// TIA Portal V18 export
FUNCTION "PLC8_910A1_CPU1214_IO_Update" : Void   // FC11010, LAD
{ S7_Optimized_Access := 'TRUE' }
VERSION : 0.1
// stored: AutoNumber false, IsIECCheckEnabled false, SetENOAutomatically false, UDAEnableTagReadback false
BEGIN

REGION Network 1: AI1 / "AI01.1.1" iw64
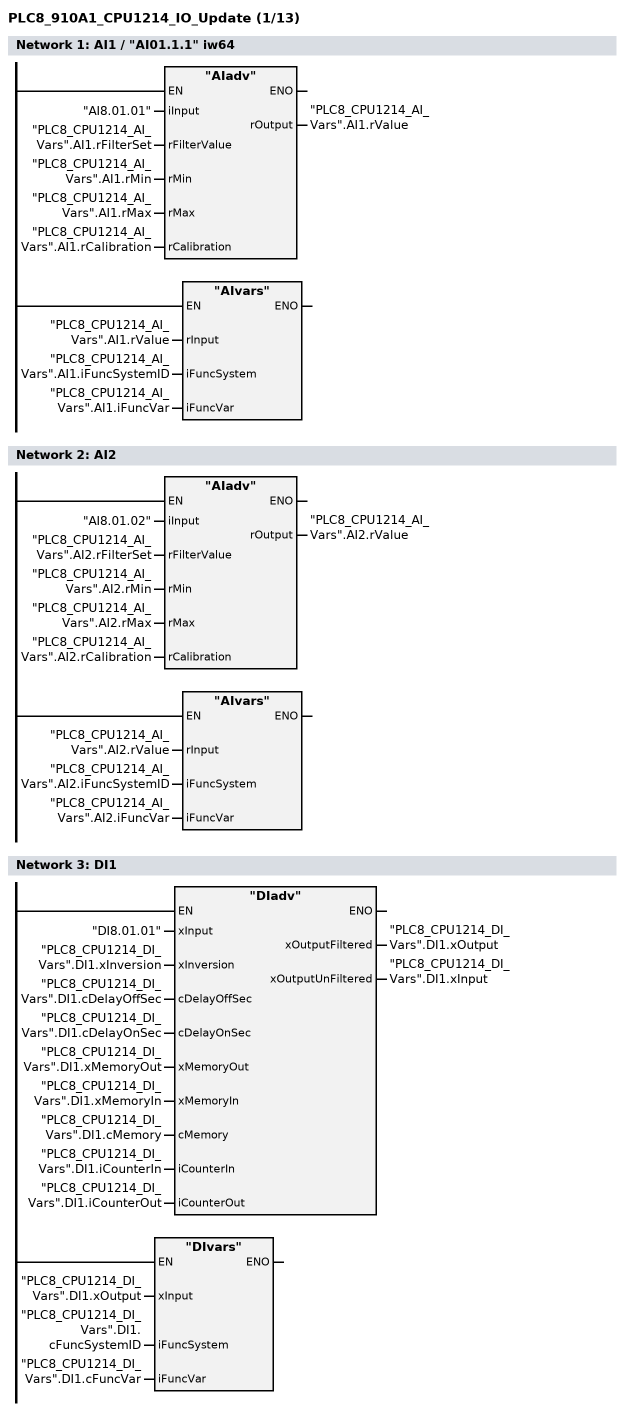
   RUNG wire#powerrail
      "AIadv"(iInput := "AI8.01.01", rFilterValue := "PLC8_CPU1214_AI_Vars".AI1.rFilterSet, rMin := "PLC8_CPU1214_AI_Vars".AI1.rMin, rMax := "PLC8_CPU1214_AI_Vars".AI1.rMax, rCalibration := "PLC8_CPU1214_AI_Vars".AI1.rCalibration, rOutput => "PLC8_CPU1214_AI_Vars".AI1.rValue)
   END_RUNG
   RUNG wire#powerrail
      "AIvars"(rInput := "PLC8_CPU1214_AI_Vars".AI1.rValue, iFuncSystem := "PLC8_CPU1214_AI_Vars".AI1.iFuncSystemID, iFuncVar := "PLC8_CPU1214_AI_Vars".AI1.iFuncVar)
   END_RUNG
   // the same network as SCL:
   "AIadv"(iInput := "AI8.01.01",
           rFilterValue := "PLC8_CPU1214_AI_Vars".AI1.rFilterSet,
           rMin := "PLC8_CPU1214_AI_Vars".AI1.rMin,
           rMax := "PLC8_CPU1214_AI_Vars".AI1.rMax,
           rCalibration := "PLC8_CPU1214_AI_Vars".AI1.rCalibration,
           rOutput => "PLC8_CPU1214_AI_Vars".AI1.rValue);
   "AIvars"(rInput := "PLC8_CPU1214_AI_Vars".AI1.rValue,
            iFuncSystem := "PLC8_CPU1214_AI_Vars".AI1.iFuncSystemID,
            iFuncVar := "PLC8_CPU1214_AI_Vars".AI1.iFuncVar);
END_REGION

REGION Network 2: AI2
   RUNG wire#powerrail
      "AIadv"(iInput := "AI8.01.02", rFilterValue := "PLC8_CPU1214_AI_Vars".AI2.rFilterSet, rMin := "PLC8_CPU1214_AI_Vars".AI2.rMin, rMax := "PLC8_CPU1214_AI_Vars".AI2.rMax, rCalibration := "PLC8_CPU1214_AI_Vars".AI2.rCalibration, rOutput => "PLC8_CPU1214_AI_Vars".AI2.rValue)
   END_RUNG
   RUNG wire#powerrail
      "AIvars"(rInput := "PLC8_CPU1214_AI_Vars".AI2.rValue, iFuncSystem := "PLC8_CPU1214_AI_Vars".AI2.iFuncSystemID, iFuncVar := "PLC8_CPU1214_AI_Vars".AI2.iFuncVar)
   END_RUNG
   // the same network as SCL:
   "AIadv"(iInput := "AI8.01.02",
           rFilterValue := "PLC8_CPU1214_AI_Vars".AI2.rFilterSet,
           rMin := "PLC8_CPU1214_AI_Vars".AI2.rMin,
           rMax := "PLC8_CPU1214_AI_Vars".AI2.rMax,
           rCalibration := "PLC8_CPU1214_AI_Vars".AI2.rCalibration,
           rOutput => "PLC8_CPU1214_AI_Vars".AI2.rValue);
   "AIvars"(rInput := "PLC8_CPU1214_AI_Vars".AI2.rValue,
            iFuncSystem := "PLC8_CPU1214_AI_Vars".AI2.iFuncSystemID,
            iFuncVar := "PLC8_CPU1214_AI_Vars".AI2.iFuncVar);
END_REGION

REGION Network 3: DI1
   RUNG wire#powerrail
      "DIadv"(xInput := "DI8.01.01", xInversion := "PLC8_CPU1214_DI_Vars".DI1.xInversion, cDelayOffSec := "PLC8_CPU1214_DI_Vars".DI1.cDelayOffSec, cDelayOnSec := "PLC8_CPU1214_DI_Vars".DI1.cDelayOnSec, xMemoryOut := "PLC8_CPU1214_DI_Vars".DI1.xMemoryOut, xMemoryIn := "PLC8_CPU1214_DI_Vars".DI1.xMemoryIn, cMemory := "PLC8_CPU1214_DI_Vars".DI1.cMemory, iCounterIn := "PLC8_CPU1214_DI_Vars".DI1.iCounterIn, iCounterOut := "PLC8_CPU1214_DI_Vars".DI1.iCounterOut, xOutputFiltered => "PLC8_CPU1214_DI_Vars".DI1.xOutput, xOutputUnFiltered => "PLC8_CPU1214_DI_Vars".DI1.xInput)
   END_RUNG
   RUNG wire#powerrail
      "DIvars"(xInput := "PLC8_CPU1214_DI_Vars".DI1.xOutput, iFuncSystem := "PLC8_CPU1214_DI_Vars".DI1.cFuncSystemID, iFuncVar := "PLC8_CPU1214_DI_Vars".DI1.cFuncVar)
   END_RUNG
   // the same network as SCL:
   "DIadv"(xInput := "DI8.01.01",
           xInversion := "PLC8_CPU1214_DI_Vars".DI1.xInversion,
           cDelayOffSec := "PLC8_CPU1214_DI_Vars".DI1.cDelayOffSec,
           cDelayOnSec := "PLC8_CPU1214_DI_Vars".DI1.cDelayOnSec,
           xMemoryOut := "PLC8_CPU1214_DI_Vars".DI1.xMemoryOut,
           xMemoryIn := "PLC8_CPU1214_DI_Vars".DI1.xMemoryIn,
           cMemory := "PLC8_CPU1214_DI_Vars".DI1.cMemory,
           iCounterIn := "PLC8_CPU1214_DI_Vars".DI1.iCounterIn,
           iCounterOut := "PLC8_CPU1214_DI_Vars".DI1.iCounterOut,
           xOutputFiltered => "PLC8_CPU1214_DI_Vars".DI1.xOutput,
           xOutputUnFiltered => "PLC8_CPU1214_DI_Vars".DI1.xInput);
   "DIvars"(xInput := "PLC8_CPU1214_DI_Vars".DI1.xOutput,
            iFuncSystem := "PLC8_CPU1214_DI_Vars".DI1.cFuncSystemID,
            iFuncVar := "PLC8_CPU1214_DI_Vars".DI1.cFuncVar);
END_REGION

REGION Network 4: DI2
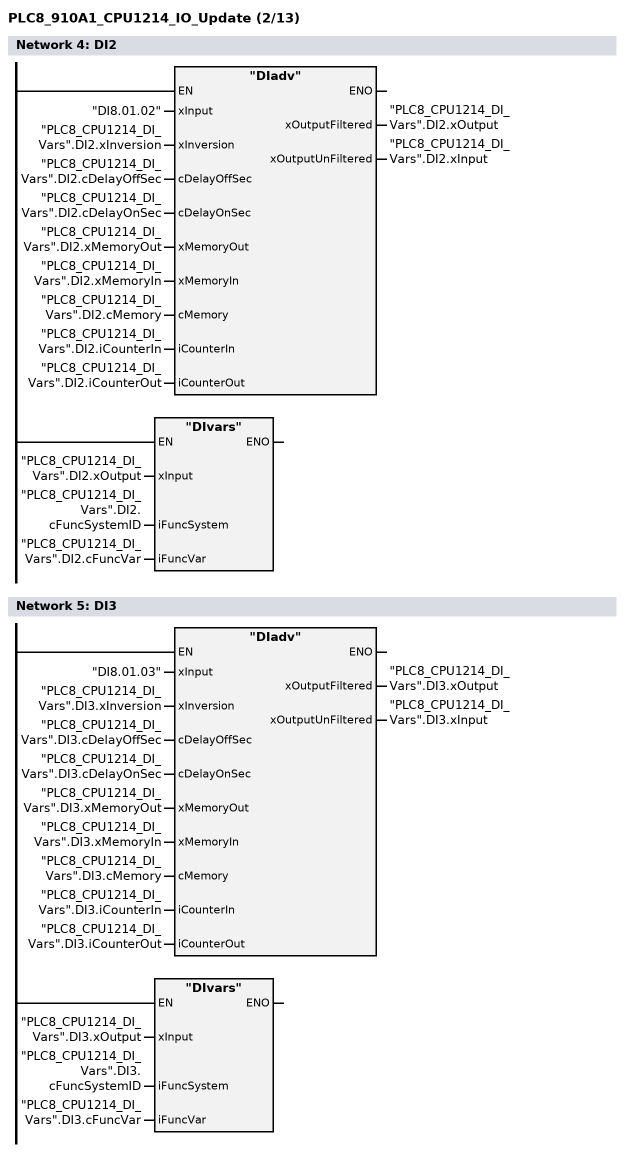
   RUNG wire#powerrail
      "DIadv"(xInput := "DI8.01.02", xInversion := "PLC8_CPU1214_DI_Vars".DI2.xInversion, cDelayOffSec := "PLC8_CPU1214_DI_Vars".DI2.cDelayOffSec, cDelayOnSec := "PLC8_CPU1214_DI_Vars".DI2.cDelayOnSec, xMemoryOut := "PLC8_CPU1214_DI_Vars".DI2.xMemoryOut, xMemoryIn := "PLC8_CPU1214_DI_Vars".DI2.xMemoryIn, cMemory := "PLC8_CPU1214_DI_Vars".DI2.cMemory, iCounterIn := "PLC8_CPU1214_DI_Vars".DI2.iCounterIn, iCounterOut := "PLC8_CPU1214_DI_Vars".DI2.iCounterOut, xOutputFiltered => "PLC8_CPU1214_DI_Vars".DI2.xOutput, xOutputUnFiltered => "PLC8_CPU1214_DI_Vars".DI2.xInput)
   END_RUNG
   RUNG wire#powerrail
      "DIvars"(xInput := "PLC8_CPU1214_DI_Vars".DI2.xOutput, iFuncSystem := "PLC8_CPU1214_DI_Vars".DI2.cFuncSystemID, iFuncVar := "PLC8_CPU1214_DI_Vars".DI2.cFuncVar)
   END_RUNG
   // the same network as SCL:
   "DIadv"(xInput := "DI8.01.02",
           xInversion := "PLC8_CPU1214_DI_Vars".DI2.xInversion,
           cDelayOffSec := "PLC8_CPU1214_DI_Vars".DI2.cDelayOffSec,
           cDelayOnSec := "PLC8_CPU1214_DI_Vars".DI2.cDelayOnSec,
           xMemoryOut := "PLC8_CPU1214_DI_Vars".DI2.xMemoryOut,
           xMemoryIn := "PLC8_CPU1214_DI_Vars".DI2.xMemoryIn,
           cMemory := "PLC8_CPU1214_DI_Vars".DI2.cMemory,
           iCounterIn := "PLC8_CPU1214_DI_Vars".DI2.iCounterIn,
           iCounterOut := "PLC8_CPU1214_DI_Vars".DI2.iCounterOut,
           xOutputFiltered => "PLC8_CPU1214_DI_Vars".DI2.xOutput,
           xOutputUnFiltered => "PLC8_CPU1214_DI_Vars".DI2.xInput);
   "DIvars"(xInput := "PLC8_CPU1214_DI_Vars".DI2.xOutput,
            iFuncSystem := "PLC8_CPU1214_DI_Vars".DI2.cFuncSystemID,
            iFuncVar := "PLC8_CPU1214_DI_Vars".DI2.cFuncVar);
END_REGION

REGION Network 5: DI3
   RUNG wire#powerrail
      "DIadv"(xInput := "DI8.01.03", xInversion := "PLC8_CPU1214_DI_Vars".DI3.xInversion, cDelayOffSec := "PLC8_CPU1214_DI_Vars".DI3.cDelayOffSec, cDelayOnSec := "PLC8_CPU1214_DI_Vars".DI3.cDelayOnSec, xMemoryOut := "PLC8_CPU1214_DI_Vars".DI3.xMemoryOut, xMemoryIn := "PLC8_CPU1214_DI_Vars".DI3.xMemoryIn, cMemory := "PLC8_CPU1214_DI_Vars".DI3.cMemory, iCounterIn := "PLC8_CPU1214_DI_Vars".DI3.iCounterIn, iCounterOut := "PLC8_CPU1214_DI_Vars".DI3.iCounterOut, xOutputFiltered => "PLC8_CPU1214_DI_Vars".DI3.xOutput, xOutputUnFiltered => "PLC8_CPU1214_DI_Vars".DI3.xInput)
   END_RUNG
   RUNG wire#powerrail
      "DIvars"(xInput := "PLC8_CPU1214_DI_Vars".DI3.xOutput, iFuncSystem := "PLC8_CPU1214_DI_Vars".DI3.cFuncSystemID, iFuncVar := "PLC8_CPU1214_DI_Vars".DI3.cFuncVar)
   END_RUNG
   // the same network as SCL:
   "DIadv"(xInput := "DI8.01.03",
           xInversion := "PLC8_CPU1214_DI_Vars".DI3.xInversion,
           cDelayOffSec := "PLC8_CPU1214_DI_Vars".DI3.cDelayOffSec,
           cDelayOnSec := "PLC8_CPU1214_DI_Vars".DI3.cDelayOnSec,
           xMemoryOut := "PLC8_CPU1214_DI_Vars".DI3.xMemoryOut,
           xMemoryIn := "PLC8_CPU1214_DI_Vars".DI3.xMemoryIn,
           cMemory := "PLC8_CPU1214_DI_Vars".DI3.cMemory,
           iCounterIn := "PLC8_CPU1214_DI_Vars".DI3.iCounterIn,
           iCounterOut := "PLC8_CPU1214_DI_Vars".DI3.iCounterOut,
           xOutputFiltered => "PLC8_CPU1214_DI_Vars".DI3.xOutput,
           xOutputUnFiltered => "PLC8_CPU1214_DI_Vars".DI3.xInput);
   "DIvars"(xInput := "PLC8_CPU1214_DI_Vars".DI3.xOutput,
            iFuncSystem := "PLC8_CPU1214_DI_Vars".DI3.cFuncSystemID,
            iFuncVar := "PLC8_CPU1214_DI_Vars".DI3.cFuncVar);
END_REGION

REGION Network 6: DI4
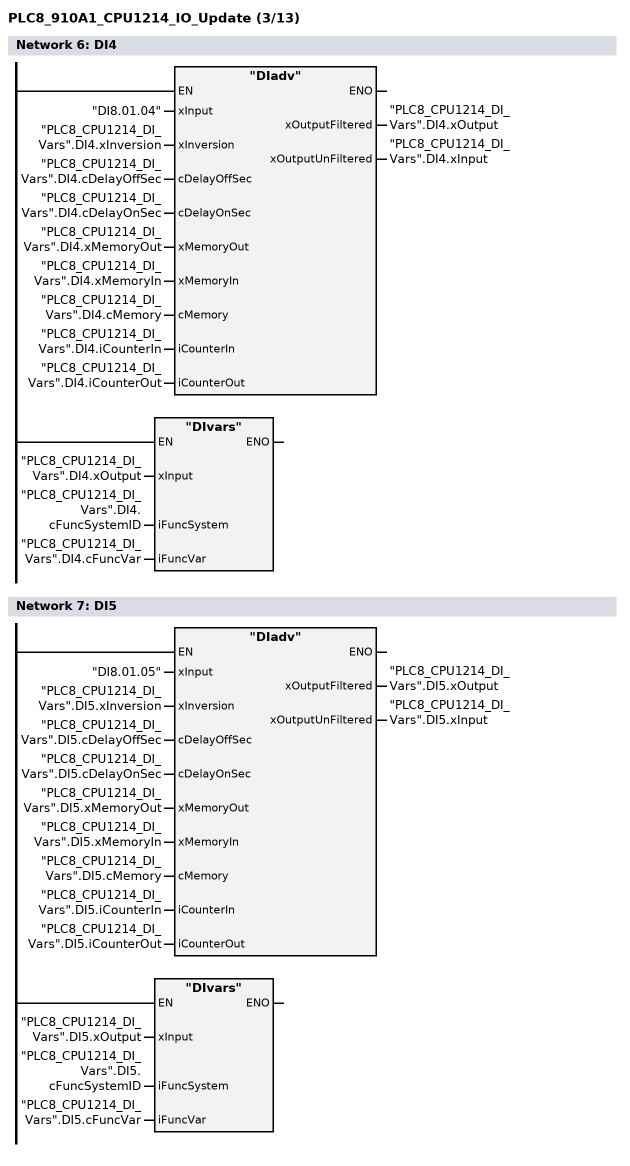
   RUNG wire#powerrail
      "DIadv"(xInput := "DI8.01.04", xInversion := "PLC8_CPU1214_DI_Vars".DI4.xInversion, cDelayOffSec := "PLC8_CPU1214_DI_Vars".DI4.cDelayOffSec, cDelayOnSec := "PLC8_CPU1214_DI_Vars".DI4.cDelayOnSec, xMemoryOut := "PLC8_CPU1214_DI_Vars".DI4.xMemoryOut, xMemoryIn := "PLC8_CPU1214_DI_Vars".DI4.xMemoryIn, cMemory := "PLC8_CPU1214_DI_Vars".DI4.cMemory, iCounterIn := "PLC8_CPU1214_DI_Vars".DI4.iCounterIn, iCounterOut := "PLC8_CPU1214_DI_Vars".DI4.iCounterOut, xOutputFiltered => "PLC8_CPU1214_DI_Vars".DI4.xOutput, xOutputUnFiltered => "PLC8_CPU1214_DI_Vars".DI4.xInput)
   END_RUNG
   RUNG wire#powerrail
      "DIvars"(xInput := "PLC8_CPU1214_DI_Vars".DI4.xOutput, iFuncSystem := "PLC8_CPU1214_DI_Vars".DI4.cFuncSystemID, iFuncVar := "PLC8_CPU1214_DI_Vars".DI4.cFuncVar)
   END_RUNG
   // the same network as SCL:
   "DIadv"(xInput := "DI8.01.04",
           xInversion := "PLC8_CPU1214_DI_Vars".DI4.xInversion,
           cDelayOffSec := "PLC8_CPU1214_DI_Vars".DI4.cDelayOffSec,
           cDelayOnSec := "PLC8_CPU1214_DI_Vars".DI4.cDelayOnSec,
           xMemoryOut := "PLC8_CPU1214_DI_Vars".DI4.xMemoryOut,
           xMemoryIn := "PLC8_CPU1214_DI_Vars".DI4.xMemoryIn,
           cMemory := "PLC8_CPU1214_DI_Vars".DI4.cMemory,
           iCounterIn := "PLC8_CPU1214_DI_Vars".DI4.iCounterIn,
           iCounterOut := "PLC8_CPU1214_DI_Vars".DI4.iCounterOut,
           xOutputFiltered => "PLC8_CPU1214_DI_Vars".DI4.xOutput,
           xOutputUnFiltered => "PLC8_CPU1214_DI_Vars".DI4.xInput);
   "DIvars"(xInput := "PLC8_CPU1214_DI_Vars".DI4.xOutput,
            iFuncSystem := "PLC8_CPU1214_DI_Vars".DI4.cFuncSystemID,
            iFuncVar := "PLC8_CPU1214_DI_Vars".DI4.cFuncVar);
END_REGION

REGION Network 7: DI5
   RUNG wire#powerrail
      "DIadv"(xInput := "DI8.01.05", xInversion := "PLC8_CPU1214_DI_Vars".DI5.xInversion, cDelayOffSec := "PLC8_CPU1214_DI_Vars".DI5.cDelayOffSec, cDelayOnSec := "PLC8_CPU1214_DI_Vars".DI5.cDelayOnSec, xMemoryOut := "PLC8_CPU1214_DI_Vars".DI5.xMemoryOut, xMemoryIn := "PLC8_CPU1214_DI_Vars".DI5.xMemoryIn, cMemory := "PLC8_CPU1214_DI_Vars".DI5.cMemory, iCounterIn := "PLC8_CPU1214_DI_Vars".DI5.iCounterIn, iCounterOut := "PLC8_CPU1214_DI_Vars".DI5.iCounterOut, xOutputFiltered => "PLC8_CPU1214_DI_Vars".DI5.xOutput, xOutputUnFiltered => "PLC8_CPU1214_DI_Vars".DI5.xInput)
   END_RUNG
   RUNG wire#powerrail
      "DIvars"(xInput := "PLC8_CPU1214_DI_Vars".DI5.xOutput, iFuncSystem := "PLC8_CPU1214_DI_Vars".DI5.cFuncSystemID, iFuncVar := "PLC8_CPU1214_DI_Vars".DI5.cFuncVar)
   END_RUNG
   // the same network as SCL:
   "DIadv"(xInput := "DI8.01.05",
           xInversion := "PLC8_CPU1214_DI_Vars".DI5.xInversion,
           cDelayOffSec := "PLC8_CPU1214_DI_Vars".DI5.cDelayOffSec,
           cDelayOnSec := "PLC8_CPU1214_DI_Vars".DI5.cDelayOnSec,
           xMemoryOut := "PLC8_CPU1214_DI_Vars".DI5.xMemoryOut,
           xMemoryIn := "PLC8_CPU1214_DI_Vars".DI5.xMemoryIn,
           cMemory := "PLC8_CPU1214_DI_Vars".DI5.cMemory,
           iCounterIn := "PLC8_CPU1214_DI_Vars".DI5.iCounterIn,
           iCounterOut := "PLC8_CPU1214_DI_Vars".DI5.iCounterOut,
           xOutputFiltered => "PLC8_CPU1214_DI_Vars".DI5.xOutput,
           xOutputUnFiltered => "PLC8_CPU1214_DI_Vars".DI5.xInput);
   "DIvars"(xInput := "PLC8_CPU1214_DI_Vars".DI5.xOutput,
            iFuncSystem := "PLC8_CPU1214_DI_Vars".DI5.cFuncSystemID,
            iFuncVar := "PLC8_CPU1214_DI_Vars".DI5.cFuncVar);
END_REGION

REGION Network 8: DI6
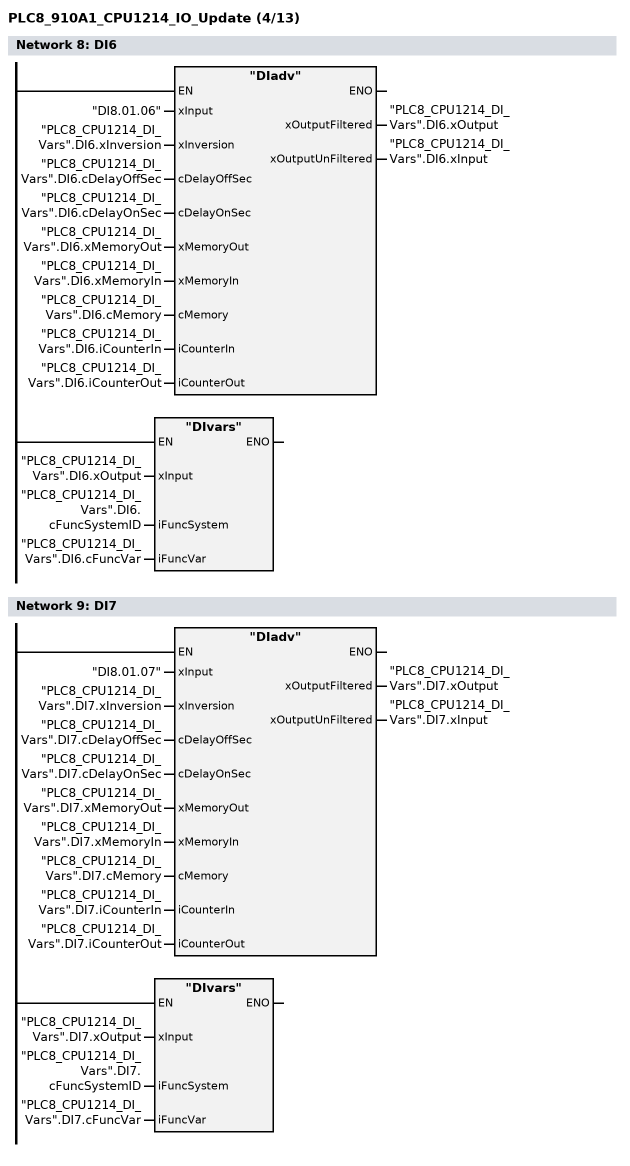
   RUNG wire#powerrail
      "DIadv"(xInput := "DI8.01.06", xInversion := "PLC8_CPU1214_DI_Vars".DI6.xInversion, cDelayOffSec := "PLC8_CPU1214_DI_Vars".DI6.cDelayOffSec, cDelayOnSec := "PLC8_CPU1214_DI_Vars".DI6.cDelayOnSec, xMemoryOut := "PLC8_CPU1214_DI_Vars".DI6.xMemoryOut, xMemoryIn := "PLC8_CPU1214_DI_Vars".DI6.xMemoryIn, cMemory := "PLC8_CPU1214_DI_Vars".DI6.cMemory, iCounterIn := "PLC8_CPU1214_DI_Vars".DI6.iCounterIn, iCounterOut := "PLC8_CPU1214_DI_Vars".DI6.iCounterOut, xOutputFiltered => "PLC8_CPU1214_DI_Vars".DI6.xOutput, xOutputUnFiltered => "PLC8_CPU1214_DI_Vars".DI6.xInput)
   END_RUNG
   RUNG wire#powerrail
      "DIvars"(xInput := "PLC8_CPU1214_DI_Vars".DI6.xOutput, iFuncSystem := "PLC8_CPU1214_DI_Vars".DI6.cFuncSystemID, iFuncVar := "PLC8_CPU1214_DI_Vars".DI6.cFuncVar)
   END_RUNG
   // the same network as SCL:
   "DIadv"(xInput := "DI8.01.06",
           xInversion := "PLC8_CPU1214_DI_Vars".DI6.xInversion,
           cDelayOffSec := "PLC8_CPU1214_DI_Vars".DI6.cDelayOffSec,
           cDelayOnSec := "PLC8_CPU1214_DI_Vars".DI6.cDelayOnSec,
           xMemoryOut := "PLC8_CPU1214_DI_Vars".DI6.xMemoryOut,
           xMemoryIn := "PLC8_CPU1214_DI_Vars".DI6.xMemoryIn,
           cMemory := "PLC8_CPU1214_DI_Vars".DI6.cMemory,
           iCounterIn := "PLC8_CPU1214_DI_Vars".DI6.iCounterIn,
           iCounterOut := "PLC8_CPU1214_DI_Vars".DI6.iCounterOut,
           xOutputFiltered => "PLC8_CPU1214_DI_Vars".DI6.xOutput,
           xOutputUnFiltered => "PLC8_CPU1214_DI_Vars".DI6.xInput);
   "DIvars"(xInput := "PLC8_CPU1214_DI_Vars".DI6.xOutput,
            iFuncSystem := "PLC8_CPU1214_DI_Vars".DI6.cFuncSystemID,
            iFuncVar := "PLC8_CPU1214_DI_Vars".DI6.cFuncVar);
END_REGION

REGION Network 9: DI7
   RUNG wire#powerrail
      "DIadv"(xInput := "DI8.01.07", xInversion := "PLC8_CPU1214_DI_Vars".DI7.xInversion, cDelayOffSec := "PLC8_CPU1214_DI_Vars".DI7.cDelayOffSec, cDelayOnSec := "PLC8_CPU1214_DI_Vars".DI7.cDelayOnSec, xMemoryOut := "PLC8_CPU1214_DI_Vars".DI7.xMemoryOut, xMemoryIn := "PLC8_CPU1214_DI_Vars".DI7.xMemoryIn, cMemory := "PLC8_CPU1214_DI_Vars".DI7.cMemory, iCounterIn := "PLC8_CPU1214_DI_Vars".DI7.iCounterIn, iCounterOut := "PLC8_CPU1214_DI_Vars".DI7.iCounterOut, xOutputFiltered => "PLC8_CPU1214_DI_Vars".DI7.xOutput, xOutputUnFiltered => "PLC8_CPU1214_DI_Vars".DI7.xInput)
   END_RUNG
   RUNG wire#powerrail
      "DIvars"(xInput := "PLC8_CPU1214_DI_Vars".DI7.xOutput, iFuncSystem := "PLC8_CPU1214_DI_Vars".DI7.cFuncSystemID, iFuncVar := "PLC8_CPU1214_DI_Vars".DI7.cFuncVar)
   END_RUNG
   // the same network as SCL:
   "DIadv"(xInput := "DI8.01.07",
           xInversion := "PLC8_CPU1214_DI_Vars".DI7.xInversion,
           cDelayOffSec := "PLC8_CPU1214_DI_Vars".DI7.cDelayOffSec,
           cDelayOnSec := "PLC8_CPU1214_DI_Vars".DI7.cDelayOnSec,
           xMemoryOut := "PLC8_CPU1214_DI_Vars".DI7.xMemoryOut,
           xMemoryIn := "PLC8_CPU1214_DI_Vars".DI7.xMemoryIn,
           cMemory := "PLC8_CPU1214_DI_Vars".DI7.cMemory,
           iCounterIn := "PLC8_CPU1214_DI_Vars".DI7.iCounterIn,
           iCounterOut := "PLC8_CPU1214_DI_Vars".DI7.iCounterOut,
           xOutputFiltered => "PLC8_CPU1214_DI_Vars".DI7.xOutput,
           xOutputUnFiltered => "PLC8_CPU1214_DI_Vars".DI7.xInput);
   "DIvars"(xInput := "PLC8_CPU1214_DI_Vars".DI7.xOutput,
            iFuncSystem := "PLC8_CPU1214_DI_Vars".DI7.cFuncSystemID,
            iFuncVar := "PLC8_CPU1214_DI_Vars".DI7.cFuncVar);
END_REGION

REGION Network 10: DI8 / DI01.1.08 EDP під охороною
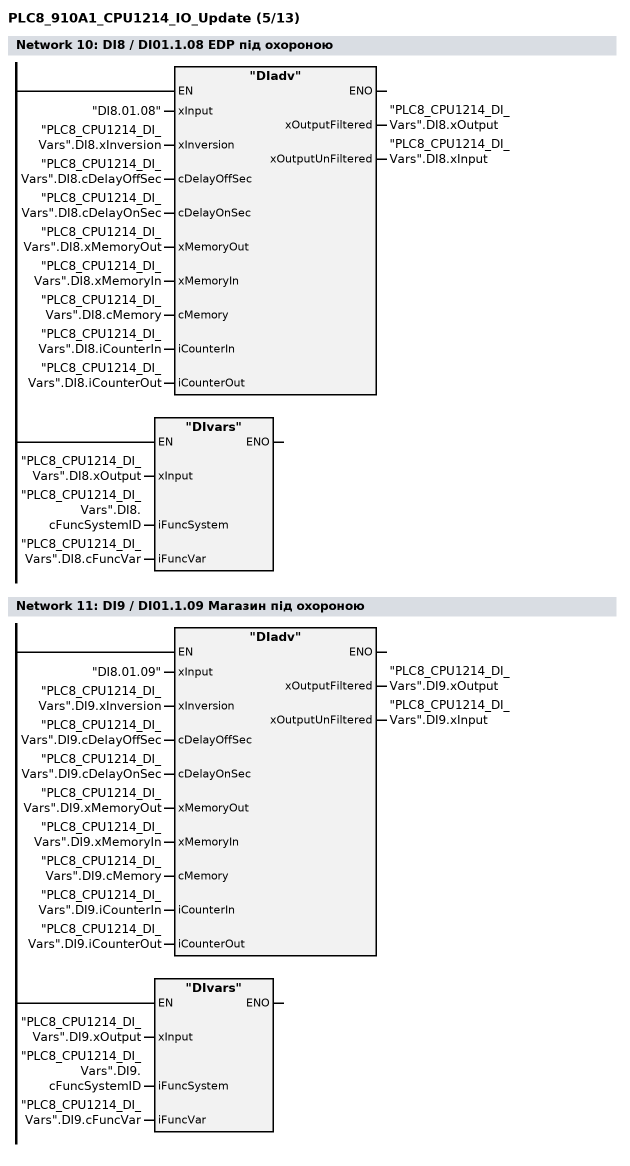
   RUNG wire#powerrail
      "DIadv"(xInput := "DI8.01.08", xInversion := "PLC8_CPU1214_DI_Vars".DI8.xInversion, cDelayOffSec := "PLC8_CPU1214_DI_Vars".DI8.cDelayOffSec, cDelayOnSec := "PLC8_CPU1214_DI_Vars".DI8.cDelayOnSec, xMemoryOut := "PLC8_CPU1214_DI_Vars".DI8.xMemoryOut, xMemoryIn := "PLC8_CPU1214_DI_Vars".DI8.xMemoryIn, cMemory := "PLC8_CPU1214_DI_Vars".DI8.cMemory, iCounterIn := "PLC8_CPU1214_DI_Vars".DI8.iCounterIn, iCounterOut := "PLC8_CPU1214_DI_Vars".DI8.iCounterOut, xOutputFiltered => "PLC8_CPU1214_DI_Vars".DI8.xOutput, xOutputUnFiltered => "PLC8_CPU1214_DI_Vars".DI8.xInput)
   END_RUNG
   RUNG wire#powerrail
      "DIvars"(xInput := "PLC8_CPU1214_DI_Vars".DI8.xOutput, iFuncSystem := "PLC8_CPU1214_DI_Vars".DI8.cFuncSystemID, iFuncVar := "PLC8_CPU1214_DI_Vars".DI8.cFuncVar)
   END_RUNG
   // the same network as SCL:
   "DIadv"(xInput := "DI8.01.08",
           xInversion := "PLC8_CPU1214_DI_Vars".DI8.xInversion,
           cDelayOffSec := "PLC8_CPU1214_DI_Vars".DI8.cDelayOffSec,
           cDelayOnSec := "PLC8_CPU1214_DI_Vars".DI8.cDelayOnSec,
           xMemoryOut := "PLC8_CPU1214_DI_Vars".DI8.xMemoryOut,
           xMemoryIn := "PLC8_CPU1214_DI_Vars".DI8.xMemoryIn,
           cMemory := "PLC8_CPU1214_DI_Vars".DI8.cMemory,
           iCounterIn := "PLC8_CPU1214_DI_Vars".DI8.iCounterIn,
           iCounterOut := "PLC8_CPU1214_DI_Vars".DI8.iCounterOut,
           xOutputFiltered => "PLC8_CPU1214_DI_Vars".DI8.xOutput,
           xOutputUnFiltered => "PLC8_CPU1214_DI_Vars".DI8.xInput);
   "DIvars"(xInput := "PLC8_CPU1214_DI_Vars".DI8.xOutput,
            iFuncSystem := "PLC8_CPU1214_DI_Vars".DI8.cFuncSystemID,
            iFuncVar := "PLC8_CPU1214_DI_Vars".DI8.cFuncVar);
END_REGION

REGION Network 11: DI9 / DI01.1.09 Магазин під охороною
   RUNG wire#powerrail
      "DIadv"(xInput := "DI8.01.09", xInversion := "PLC8_CPU1214_DI_Vars".DI9.xInversion, cDelayOffSec := "PLC8_CPU1214_DI_Vars".DI9.cDelayOffSec, cDelayOnSec := "PLC8_CPU1214_DI_Vars".DI9.cDelayOnSec, xMemoryOut := "PLC8_CPU1214_DI_Vars".DI9.xMemoryOut, xMemoryIn := "PLC8_CPU1214_DI_Vars".DI9.xMemoryIn, cMemory := "PLC8_CPU1214_DI_Vars".DI9.cMemory, iCounterIn := "PLC8_CPU1214_DI_Vars".DI9.iCounterIn, iCounterOut := "PLC8_CPU1214_DI_Vars".DI9.iCounterOut, xOutputFiltered => "PLC8_CPU1214_DI_Vars".DI9.xOutput, xOutputUnFiltered => "PLC8_CPU1214_DI_Vars".DI9.xInput)
   END_RUNG
   RUNG wire#powerrail
      "DIvars"(xInput := "PLC8_CPU1214_DI_Vars".DI9.xOutput, iFuncSystem := "PLC8_CPU1214_DI_Vars".DI9.cFuncSystemID, iFuncVar := "PLC8_CPU1214_DI_Vars".DI9.cFuncVar)
   END_RUNG
   // the same network as SCL:
   "DIadv"(xInput := "DI8.01.09",
           xInversion := "PLC8_CPU1214_DI_Vars".DI9.xInversion,
           cDelayOffSec := "PLC8_CPU1214_DI_Vars".DI9.cDelayOffSec,
           cDelayOnSec := "PLC8_CPU1214_DI_Vars".DI9.cDelayOnSec,
           xMemoryOut := "PLC8_CPU1214_DI_Vars".DI9.xMemoryOut,
           xMemoryIn := "PLC8_CPU1214_DI_Vars".DI9.xMemoryIn,
           cMemory := "PLC8_CPU1214_DI_Vars".DI9.cMemory,
           iCounterIn := "PLC8_CPU1214_DI_Vars".DI9.iCounterIn,
           iCounterOut := "PLC8_CPU1214_DI_Vars".DI9.iCounterOut,
           xOutputFiltered => "PLC8_CPU1214_DI_Vars".DI9.xOutput,
           xOutputUnFiltered => "PLC8_CPU1214_DI_Vars".DI9.xInput);
   "DIvars"(xInput := "PLC8_CPU1214_DI_Vars".DI9.xOutput,
            iFuncSystem := "PLC8_CPU1214_DI_Vars".DI9.cFuncSystemID,
            iFuncVar := "PLC8_CPU1214_DI_Vars".DI9.cFuncVar);
END_REGION

REGION Network 12: DI10 / DI01.1.10 Аварійний рівень загазованості
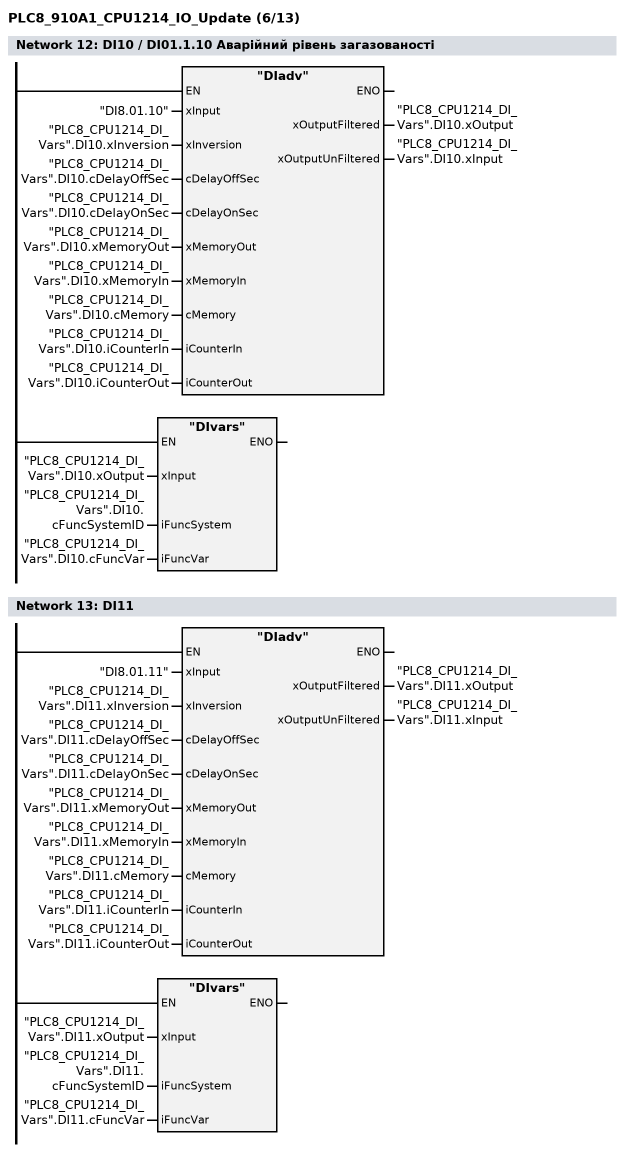
   RUNG wire#powerrail
      "DIadv"(xInput := "DI8.01.10", xInversion := "PLC8_CPU1214_DI_Vars".DI10.xInversion, cDelayOffSec := "PLC8_CPU1214_DI_Vars".DI10.cDelayOffSec, cDelayOnSec := "PLC8_CPU1214_DI_Vars".DI10.cDelayOnSec, xMemoryOut := "PLC8_CPU1214_DI_Vars".DI10.xMemoryOut, xMemoryIn := "PLC8_CPU1214_DI_Vars".DI10.xMemoryIn, cMemory := "PLC8_CPU1214_DI_Vars".DI10.cMemory, iCounterIn := "PLC8_CPU1214_DI_Vars".DI10.iCounterIn, iCounterOut := "PLC8_CPU1214_DI_Vars".DI10.iCounterOut, xOutputFiltered => "PLC8_CPU1214_DI_Vars".DI10.xOutput, xOutputUnFiltered => "PLC8_CPU1214_DI_Vars".DI10.xInput)
   END_RUNG
   RUNG wire#powerrail
      "DIvars"(xInput := "PLC8_CPU1214_DI_Vars".DI10.xOutput, iFuncSystem := "PLC8_CPU1214_DI_Vars".DI10.cFuncSystemID, iFuncVar := "PLC8_CPU1214_DI_Vars".DI10.cFuncVar)
   END_RUNG
   // the same network as SCL:
   "DIadv"(xInput := "DI8.01.10",
           xInversion := "PLC8_CPU1214_DI_Vars".DI10.xInversion,
           cDelayOffSec := "PLC8_CPU1214_DI_Vars".DI10.cDelayOffSec,
           cDelayOnSec := "PLC8_CPU1214_DI_Vars".DI10.cDelayOnSec,
           xMemoryOut := "PLC8_CPU1214_DI_Vars".DI10.xMemoryOut,
           xMemoryIn := "PLC8_CPU1214_DI_Vars".DI10.xMemoryIn,
           cMemory := "PLC8_CPU1214_DI_Vars".DI10.cMemory,
           iCounterIn := "PLC8_CPU1214_DI_Vars".DI10.iCounterIn,
           iCounterOut := "PLC8_CPU1214_DI_Vars".DI10.iCounterOut,
           xOutputFiltered => "PLC8_CPU1214_DI_Vars".DI10.xOutput,
           xOutputUnFiltered => "PLC8_CPU1214_DI_Vars".DI10.xInput);
   "DIvars"(xInput := "PLC8_CPU1214_DI_Vars".DI10.xOutput,
            iFuncSystem := "PLC8_CPU1214_DI_Vars".DI10.cFuncSystemID,
            iFuncVar := "PLC8_CPU1214_DI_Vars".DI10.cFuncVar);
END_REGION

REGION Network 13: DI11
   RUNG wire#powerrail
      "DIadv"(xInput := "DI8.01.11", xInversion := "PLC8_CPU1214_DI_Vars".DI11.xInversion, cDelayOffSec := "PLC8_CPU1214_DI_Vars".DI11.cDelayOffSec, cDelayOnSec := "PLC8_CPU1214_DI_Vars".DI11.cDelayOnSec, xMemoryOut := "PLC8_CPU1214_DI_Vars".DI11.xMemoryOut, xMemoryIn := "PLC8_CPU1214_DI_Vars".DI11.xMemoryIn, cMemory := "PLC8_CPU1214_DI_Vars".DI11.cMemory, iCounterIn := "PLC8_CPU1214_DI_Vars".DI11.iCounterIn, iCounterOut := "PLC8_CPU1214_DI_Vars".DI11.iCounterOut, xOutputFiltered => "PLC8_CPU1214_DI_Vars".DI11.xOutput, xOutputUnFiltered => "PLC8_CPU1214_DI_Vars".DI11.xInput)
   END_RUNG
   RUNG wire#powerrail
      "DIvars"(xInput := "PLC8_CPU1214_DI_Vars".DI11.xOutput, iFuncSystem := "PLC8_CPU1214_DI_Vars".DI11.cFuncSystemID, iFuncVar := "PLC8_CPU1214_DI_Vars".DI11.cFuncVar)
   END_RUNG
   // the same network as SCL:
   "DIadv"(xInput := "DI8.01.11",
           xInversion := "PLC8_CPU1214_DI_Vars".DI11.xInversion,
           cDelayOffSec := "PLC8_CPU1214_DI_Vars".DI11.cDelayOffSec,
           cDelayOnSec := "PLC8_CPU1214_DI_Vars".DI11.cDelayOnSec,
           xMemoryOut := "PLC8_CPU1214_DI_Vars".DI11.xMemoryOut,
           xMemoryIn := "PLC8_CPU1214_DI_Vars".DI11.xMemoryIn,
           cMemory := "PLC8_CPU1214_DI_Vars".DI11.cMemory,
           iCounterIn := "PLC8_CPU1214_DI_Vars".DI11.iCounterIn,
           iCounterOut := "PLC8_CPU1214_DI_Vars".DI11.iCounterOut,
           xOutputFiltered => "PLC8_CPU1214_DI_Vars".DI11.xOutput,
           xOutputUnFiltered => "PLC8_CPU1214_DI_Vars".DI11.xInput);
   "DIvars"(xInput := "PLC8_CPU1214_DI_Vars".DI11.xOutput,
            iFuncSystem := "PLC8_CPU1214_DI_Vars".DI11.cFuncSystemID,
            iFuncVar := "PLC8_CPU1214_DI_Vars".DI11.cFuncVar);
END_REGION

REGION Network 14: DI12
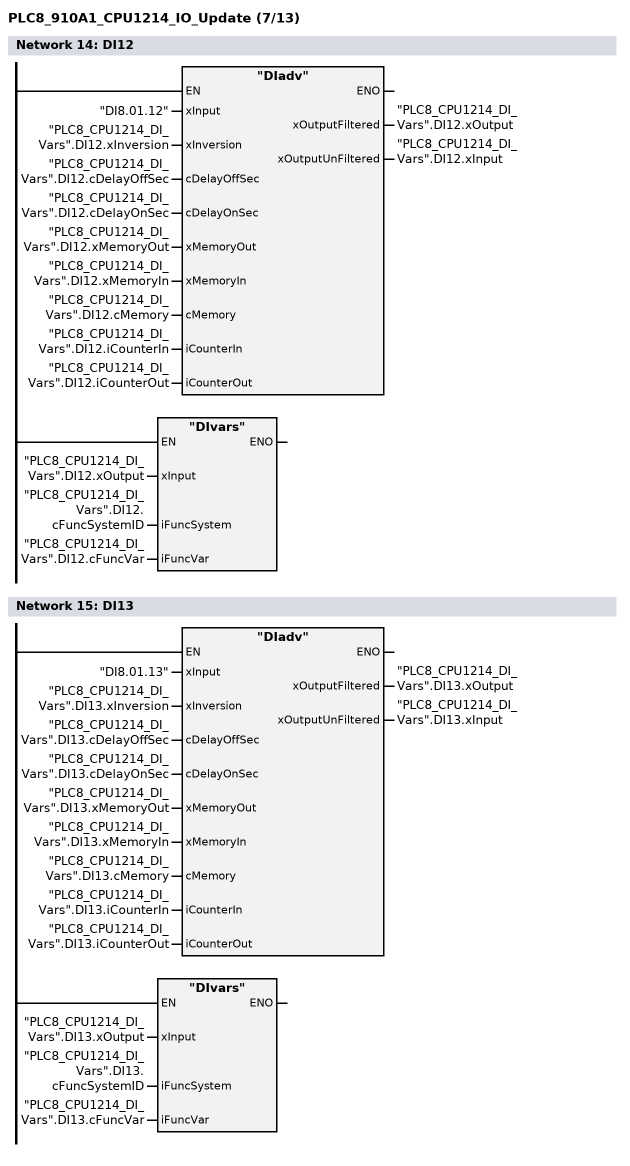
   RUNG wire#powerrail
      "DIadv"(xInput := "DI8.01.12", xInversion := "PLC8_CPU1214_DI_Vars".DI12.xInversion, cDelayOffSec := "PLC8_CPU1214_DI_Vars".DI12.cDelayOffSec, cDelayOnSec := "PLC8_CPU1214_DI_Vars".DI12.cDelayOnSec, xMemoryOut := "PLC8_CPU1214_DI_Vars".DI12.xMemoryOut, xMemoryIn := "PLC8_CPU1214_DI_Vars".DI12.xMemoryIn, cMemory := "PLC8_CPU1214_DI_Vars".DI12.cMemory, iCounterIn := "PLC8_CPU1214_DI_Vars".DI12.iCounterIn, iCounterOut := "PLC8_CPU1214_DI_Vars".DI12.iCounterOut, xOutputFiltered => "PLC8_CPU1214_DI_Vars".DI12.xOutput, xOutputUnFiltered => "PLC8_CPU1214_DI_Vars".DI12.xInput)
   END_RUNG
   RUNG wire#powerrail
      "DIvars"(xInput := "PLC8_CPU1214_DI_Vars".DI12.xOutput, iFuncSystem := "PLC8_CPU1214_DI_Vars".DI12.cFuncSystemID, iFuncVar := "PLC8_CPU1214_DI_Vars".DI12.cFuncVar)
   END_RUNG
   // the same network as SCL:
   "DIadv"(xInput := "DI8.01.12",
           xInversion := "PLC8_CPU1214_DI_Vars".DI12.xInversion,
           cDelayOffSec := "PLC8_CPU1214_DI_Vars".DI12.cDelayOffSec,
           cDelayOnSec := "PLC8_CPU1214_DI_Vars".DI12.cDelayOnSec,
           xMemoryOut := "PLC8_CPU1214_DI_Vars".DI12.xMemoryOut,
           xMemoryIn := "PLC8_CPU1214_DI_Vars".DI12.xMemoryIn,
           cMemory := "PLC8_CPU1214_DI_Vars".DI12.cMemory,
           iCounterIn := "PLC8_CPU1214_DI_Vars".DI12.iCounterIn,
           iCounterOut := "PLC8_CPU1214_DI_Vars".DI12.iCounterOut,
           xOutputFiltered => "PLC8_CPU1214_DI_Vars".DI12.xOutput,
           xOutputUnFiltered => "PLC8_CPU1214_DI_Vars".DI12.xInput);
   "DIvars"(xInput := "PLC8_CPU1214_DI_Vars".DI12.xOutput,
            iFuncSystem := "PLC8_CPU1214_DI_Vars".DI12.cFuncSystemID,
            iFuncVar := "PLC8_CPU1214_DI_Vars".DI12.cFuncVar);
END_REGION

REGION Network 15: DI13
   RUNG wire#powerrail
      "DIadv"(xInput := "DI8.01.13", xInversion := "PLC8_CPU1214_DI_Vars".DI13.xInversion, cDelayOffSec := "PLC8_CPU1214_DI_Vars".DI13.cDelayOffSec, cDelayOnSec := "PLC8_CPU1214_DI_Vars".DI13.cDelayOnSec, xMemoryOut := "PLC8_CPU1214_DI_Vars".DI13.xMemoryOut, xMemoryIn := "PLC8_CPU1214_DI_Vars".DI13.xMemoryIn, cMemory := "PLC8_CPU1214_DI_Vars".DI13.cMemory, iCounterIn := "PLC8_CPU1214_DI_Vars".DI13.iCounterIn, iCounterOut := "PLC8_CPU1214_DI_Vars".DI13.iCounterOut, xOutputFiltered => "PLC8_CPU1214_DI_Vars".DI13.xOutput, xOutputUnFiltered => "PLC8_CPU1214_DI_Vars".DI13.xInput)
   END_RUNG
   RUNG wire#powerrail
      "DIvars"(xInput := "PLC8_CPU1214_DI_Vars".DI13.xOutput, iFuncSystem := "PLC8_CPU1214_DI_Vars".DI13.cFuncSystemID, iFuncVar := "PLC8_CPU1214_DI_Vars".DI13.cFuncVar)
   END_RUNG
   // the same network as SCL:
   "DIadv"(xInput := "DI8.01.13",
           xInversion := "PLC8_CPU1214_DI_Vars".DI13.xInversion,
           cDelayOffSec := "PLC8_CPU1214_DI_Vars".DI13.cDelayOffSec,
           cDelayOnSec := "PLC8_CPU1214_DI_Vars".DI13.cDelayOnSec,
           xMemoryOut := "PLC8_CPU1214_DI_Vars".DI13.xMemoryOut,
           xMemoryIn := "PLC8_CPU1214_DI_Vars".DI13.xMemoryIn,
           cMemory := "PLC8_CPU1214_DI_Vars".DI13.cMemory,
           iCounterIn := "PLC8_CPU1214_DI_Vars".DI13.iCounterIn,
           iCounterOut := "PLC8_CPU1214_DI_Vars".DI13.iCounterOut,
           xOutputFiltered => "PLC8_CPU1214_DI_Vars".DI13.xOutput,
           xOutputUnFiltered => "PLC8_CPU1214_DI_Vars".DI13.xInput);
   "DIvars"(xInput := "PLC8_CPU1214_DI_Vars".DI13.xOutput,
            iFuncSystem := "PLC8_CPU1214_DI_Vars".DI13.cFuncSystemID,
            iFuncVar := "PLC8_CPU1214_DI_Vars".DI13.cFuncVar);
END_REGION

REGION Network 16: DI14 / DI01.1.14 Спрацювання охоронної сигналізації
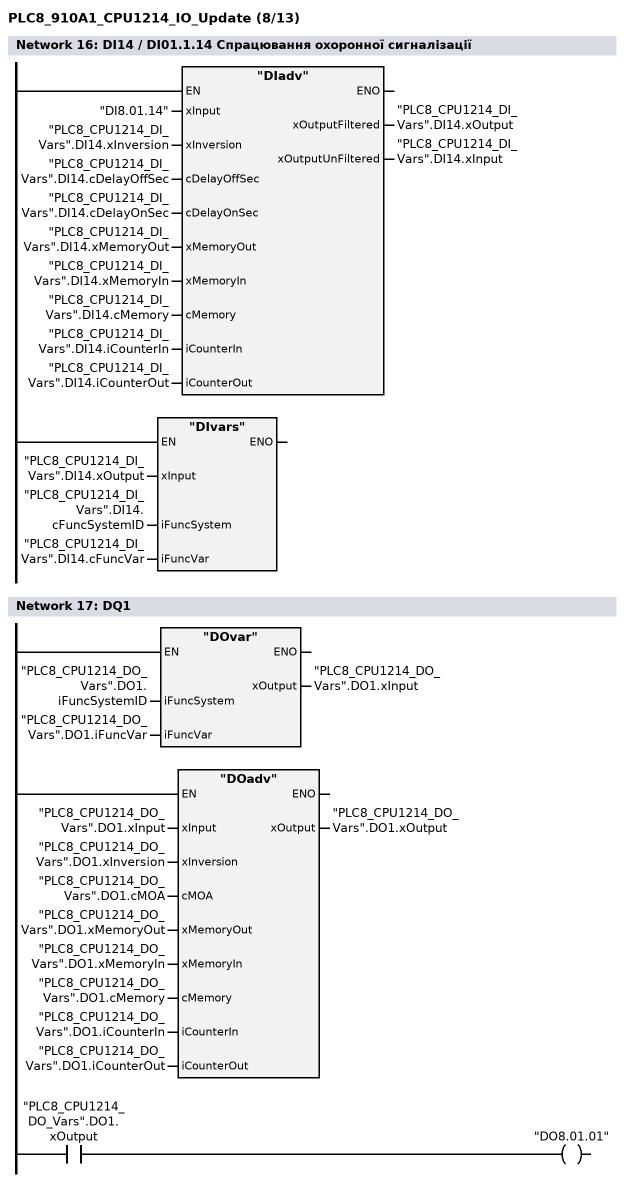
   RUNG wire#powerrail
      "DIadv"(xInput := "DI8.01.14", xInversion := "PLC8_CPU1214_DI_Vars".DI14.xInversion, cDelayOffSec := "PLC8_CPU1214_DI_Vars".DI14.cDelayOffSec, cDelayOnSec := "PLC8_CPU1214_DI_Vars".DI14.cDelayOnSec, xMemoryOut := "PLC8_CPU1214_DI_Vars".DI14.xMemoryOut, xMemoryIn := "PLC8_CPU1214_DI_Vars".DI14.xMemoryIn, cMemory := "PLC8_CPU1214_DI_Vars".DI14.cMemory, iCounterIn := "PLC8_CPU1214_DI_Vars".DI14.iCounterIn, iCounterOut := "PLC8_CPU1214_DI_Vars".DI14.iCounterOut, xOutputFiltered => "PLC8_CPU1214_DI_Vars".DI14.xOutput, xOutputUnFiltered => "PLC8_CPU1214_DI_Vars".DI14.xInput)
   END_RUNG
   RUNG wire#powerrail
      "DIvars"(xInput := "PLC8_CPU1214_DI_Vars".DI14.xOutput, iFuncSystem := "PLC8_CPU1214_DI_Vars".DI14.cFuncSystemID, iFuncVar := "PLC8_CPU1214_DI_Vars".DI14.cFuncVar)
   END_RUNG
   // the same network as SCL:
   "DIadv"(xInput := "DI8.01.14",
           xInversion := "PLC8_CPU1214_DI_Vars".DI14.xInversion,
           cDelayOffSec := "PLC8_CPU1214_DI_Vars".DI14.cDelayOffSec,
           cDelayOnSec := "PLC8_CPU1214_DI_Vars".DI14.cDelayOnSec,
           xMemoryOut := "PLC8_CPU1214_DI_Vars".DI14.xMemoryOut,
           xMemoryIn := "PLC8_CPU1214_DI_Vars".DI14.xMemoryIn,
           cMemory := "PLC8_CPU1214_DI_Vars".DI14.cMemory,
           iCounterIn := "PLC8_CPU1214_DI_Vars".DI14.iCounterIn,
           iCounterOut := "PLC8_CPU1214_DI_Vars".DI14.iCounterOut,
           xOutputFiltered => "PLC8_CPU1214_DI_Vars".DI14.xOutput,
           xOutputUnFiltered => "PLC8_CPU1214_DI_Vars".DI14.xInput);
   "DIvars"(xInput := "PLC8_CPU1214_DI_Vars".DI14.xOutput,
            iFuncSystem := "PLC8_CPU1214_DI_Vars".DI14.cFuncSystemID,
            iFuncVar := "PLC8_CPU1214_DI_Vars".DI14.cFuncVar);
END_REGION

REGION Network 17: DQ1
   RUNG wire#powerrail
      "DOvar"(iFuncSystem := "PLC8_CPU1214_DO_Vars".DO1.iFuncSystemID, iFuncVar := "PLC8_CPU1214_DO_Vars".DO1.iFuncVar, xOutput => "PLC8_CPU1214_DO_Vars".DO1.xInput)
   END_RUNG
   RUNG wire#powerrail
      "DOadv"(xInput := "PLC8_CPU1214_DO_Vars".DO1.xInput, xInversion := "PLC8_CPU1214_DO_Vars".DO1.xInversion, cMOA := "PLC8_CPU1214_DO_Vars".DO1.cMOA, xMemoryOut := "PLC8_CPU1214_DO_Vars".DO1.xMemoryOut, xMemoryIn := "PLC8_CPU1214_DO_Vars".DO1.xMemoryIn, cMemory := "PLC8_CPU1214_DO_Vars".DO1.cMemory, iCounterIn := "PLC8_CPU1214_DO_Vars".DO1.iCounterIn, iCounterOut := "PLC8_CPU1214_DO_Vars".DO1.iCounterOut, xOutput => "PLC8_CPU1214_DO_Vars".DO1.xOutput)
   END_RUNG
   RUNG wire#powerrail
      Contact( "PLC8_CPU1214_DO_Vars".DO1.xOutput )
      Coil( "DO8.01.01" )
   END_RUNG
   // the same network as SCL:
   "DOvar"(iFuncSystem := "PLC8_CPU1214_DO_Vars".DO1.iFuncSystemID,
           iFuncVar := "PLC8_CPU1214_DO_Vars".DO1.iFuncVar,
           xOutput => "PLC8_CPU1214_DO_Vars".DO1.xInput);
   "DOadv"(xInput := "PLC8_CPU1214_DO_Vars".DO1.xInput,
           xInversion := "PLC8_CPU1214_DO_Vars".DO1.xInversion,
           cMOA := "PLC8_CPU1214_DO_Vars".DO1.cMOA,
           xMemoryOut := "PLC8_CPU1214_DO_Vars".DO1.xMemoryOut,
           xMemoryIn := "PLC8_CPU1214_DO_Vars".DO1.xMemoryIn,
           cMemory := "PLC8_CPU1214_DO_Vars".DO1.cMemory,
           iCounterIn := "PLC8_CPU1214_DO_Vars".DO1.iCounterIn,
           iCounterOut := "PLC8_CPU1214_DO_Vars".DO1.iCounterOut,
           xOutput => "PLC8_CPU1214_DO_Vars".DO1.xOutput);
   "DO8.01.01" := "PLC8_CPU1214_DO_Vars".DO1.xOutput;
END_REGION

REGION Network 18: DQ2
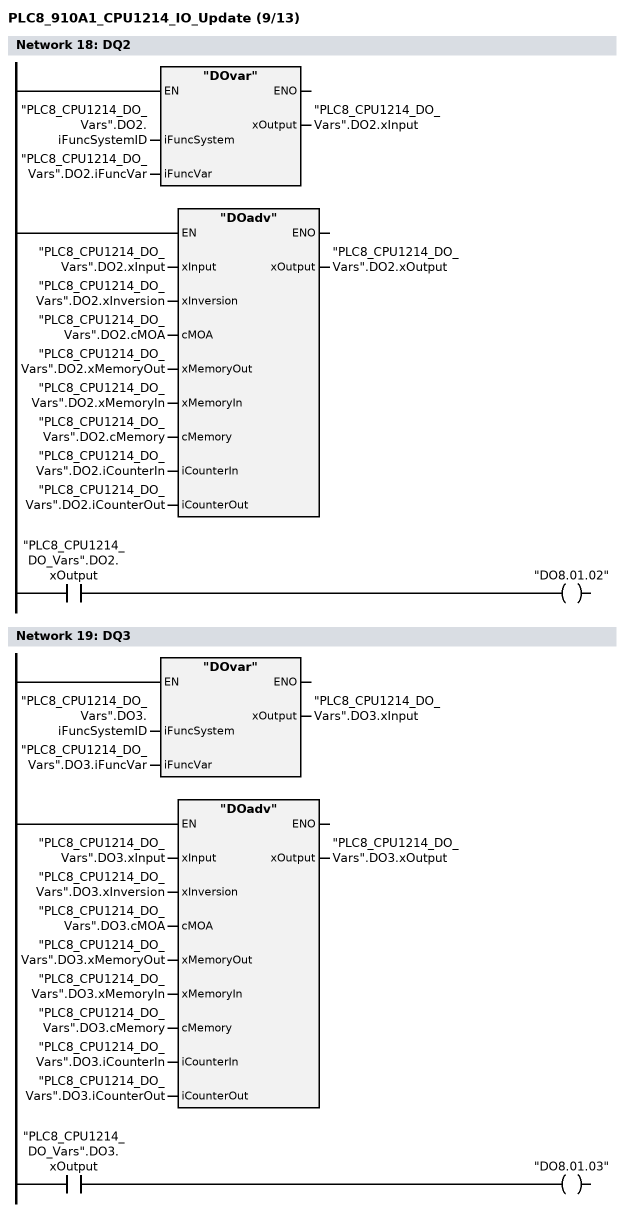
   RUNG wire#powerrail
      "DOvar"(iFuncSystem := "PLC8_CPU1214_DO_Vars".DO2.iFuncSystemID, iFuncVar := "PLC8_CPU1214_DO_Vars".DO2.iFuncVar, xOutput => "PLC8_CPU1214_DO_Vars".DO2.xInput)
   END_RUNG
   RUNG wire#powerrail
      "DOadv"(xInput := "PLC8_CPU1214_DO_Vars".DO2.xInput, xInversion := "PLC8_CPU1214_DO_Vars".DO2.xInversion, cMOA := "PLC8_CPU1214_DO_Vars".DO2.cMOA, xMemoryOut := "PLC8_CPU1214_DO_Vars".DO2.xMemoryOut, xMemoryIn := "PLC8_CPU1214_DO_Vars".DO2.xMemoryIn, cMemory := "PLC8_CPU1214_DO_Vars".DO2.cMemory, iCounterIn := "PLC8_CPU1214_DO_Vars".DO2.iCounterIn, iCounterOut := "PLC8_CPU1214_DO_Vars".DO2.iCounterOut, xOutput => "PLC8_CPU1214_DO_Vars".DO2.xOutput)
   END_RUNG
   RUNG wire#powerrail
      Contact( "PLC8_CPU1214_DO_Vars".DO2.xOutput )
      Coil( "DO8.01.02" )
   END_RUNG
   // the same network as SCL:
   "DOvar"(iFuncSystem := "PLC8_CPU1214_DO_Vars".DO2.iFuncSystemID,
           iFuncVar := "PLC8_CPU1214_DO_Vars".DO2.iFuncVar,
           xOutput => "PLC8_CPU1214_DO_Vars".DO2.xInput);
   "DOadv"(xInput := "PLC8_CPU1214_DO_Vars".DO2.xInput,
           xInversion := "PLC8_CPU1214_DO_Vars".DO2.xInversion,
           cMOA := "PLC8_CPU1214_DO_Vars".DO2.cMOA,
           xMemoryOut := "PLC8_CPU1214_DO_Vars".DO2.xMemoryOut,
           xMemoryIn := "PLC8_CPU1214_DO_Vars".DO2.xMemoryIn,
           cMemory := "PLC8_CPU1214_DO_Vars".DO2.cMemory,
           iCounterIn := "PLC8_CPU1214_DO_Vars".DO2.iCounterIn,
           iCounterOut := "PLC8_CPU1214_DO_Vars".DO2.iCounterOut,
           xOutput => "PLC8_CPU1214_DO_Vars".DO2.xOutput);
   "DO8.01.02" := "PLC8_CPU1214_DO_Vars".DO2.xOutput;
END_REGION

REGION Network 19: DQ3
   RUNG wire#powerrail
      "DOvar"(iFuncSystem := "PLC8_CPU1214_DO_Vars".DO3.iFuncSystemID, iFuncVar := "PLC8_CPU1214_DO_Vars".DO3.iFuncVar, xOutput => "PLC8_CPU1214_DO_Vars".DO3.xInput)
   END_RUNG
   RUNG wire#powerrail
      "DOadv"(xInput := "PLC8_CPU1214_DO_Vars".DO3.xInput, xInversion := "PLC8_CPU1214_DO_Vars".DO3.xInversion, cMOA := "PLC8_CPU1214_DO_Vars".DO3.cMOA, xMemoryOut := "PLC8_CPU1214_DO_Vars".DO3.xMemoryOut, xMemoryIn := "PLC8_CPU1214_DO_Vars".DO3.xMemoryIn, cMemory := "PLC8_CPU1214_DO_Vars".DO3.cMemory, iCounterIn := "PLC8_CPU1214_DO_Vars".DO3.iCounterIn, iCounterOut := "PLC8_CPU1214_DO_Vars".DO3.iCounterOut, xOutput => "PLC8_CPU1214_DO_Vars".DO3.xOutput)
   END_RUNG
   RUNG wire#powerrail
      Contact( "PLC8_CPU1214_DO_Vars".DO3.xOutput )
      Coil( "DO8.01.03" )
   END_RUNG
   // the same network as SCL:
   "DOvar"(iFuncSystem := "PLC8_CPU1214_DO_Vars".DO3.iFuncSystemID,
           iFuncVar := "PLC8_CPU1214_DO_Vars".DO3.iFuncVar,
           xOutput => "PLC8_CPU1214_DO_Vars".DO3.xInput);
   "DOadv"(xInput := "PLC8_CPU1214_DO_Vars".DO3.xInput,
           xInversion := "PLC8_CPU1214_DO_Vars".DO3.xInversion,
           cMOA := "PLC8_CPU1214_DO_Vars".DO3.cMOA,
           xMemoryOut := "PLC8_CPU1214_DO_Vars".DO3.xMemoryOut,
           xMemoryIn := "PLC8_CPU1214_DO_Vars".DO3.xMemoryIn,
           cMemory := "PLC8_CPU1214_DO_Vars".DO3.cMemory,
           iCounterIn := "PLC8_CPU1214_DO_Vars".DO3.iCounterIn,
           iCounterOut := "PLC8_CPU1214_DO_Vars".DO3.iCounterOut,
           xOutput => "PLC8_CPU1214_DO_Vars".DO3.xOutput);
   "DO8.01.03" := "PLC8_CPU1214_DO_Vars".DO3.xOutput;
END_REGION

REGION Network 20: DQ4
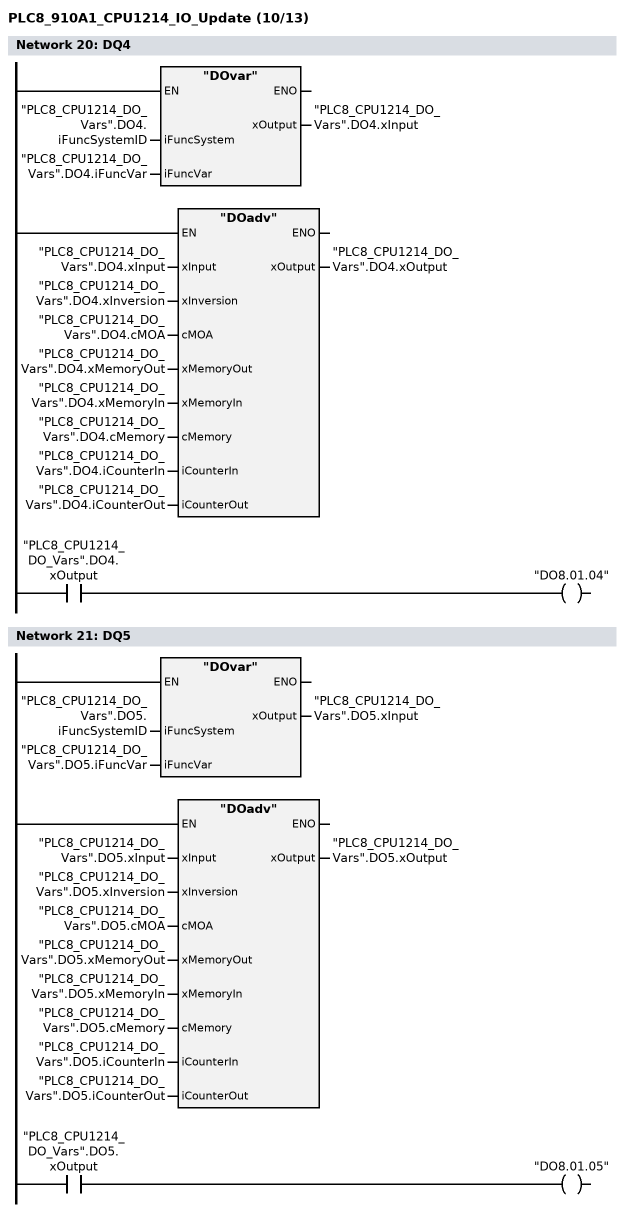
   RUNG wire#powerrail
      "DOvar"(iFuncSystem := "PLC8_CPU1214_DO_Vars".DO4.iFuncSystemID, iFuncVar := "PLC8_CPU1214_DO_Vars".DO4.iFuncVar, xOutput => "PLC8_CPU1214_DO_Vars".DO4.xInput)
   END_RUNG
   RUNG wire#powerrail
      "DOadv"(xInput := "PLC8_CPU1214_DO_Vars".DO4.xInput, xInversion := "PLC8_CPU1214_DO_Vars".DO4.xInversion, cMOA := "PLC8_CPU1214_DO_Vars".DO4.cMOA, xMemoryOut := "PLC8_CPU1214_DO_Vars".DO4.xMemoryOut, xMemoryIn := "PLC8_CPU1214_DO_Vars".DO4.xMemoryIn, cMemory := "PLC8_CPU1214_DO_Vars".DO4.cMemory, iCounterIn := "PLC8_CPU1214_DO_Vars".DO4.iCounterIn, iCounterOut := "PLC8_CPU1214_DO_Vars".DO4.iCounterOut, xOutput => "PLC8_CPU1214_DO_Vars".DO4.xOutput)
   END_RUNG
   RUNG wire#powerrail
      Contact( "PLC8_CPU1214_DO_Vars".DO4.xOutput )
      Coil( "DO8.01.04" )
   END_RUNG
   // the same network as SCL:
   "DOvar"(iFuncSystem := "PLC8_CPU1214_DO_Vars".DO4.iFuncSystemID,
           iFuncVar := "PLC8_CPU1214_DO_Vars".DO4.iFuncVar,
           xOutput => "PLC8_CPU1214_DO_Vars".DO4.xInput);
   "DOadv"(xInput := "PLC8_CPU1214_DO_Vars".DO4.xInput,
           xInversion := "PLC8_CPU1214_DO_Vars".DO4.xInversion,
           cMOA := "PLC8_CPU1214_DO_Vars".DO4.cMOA,
           xMemoryOut := "PLC8_CPU1214_DO_Vars".DO4.xMemoryOut,
           xMemoryIn := "PLC8_CPU1214_DO_Vars".DO4.xMemoryIn,
           cMemory := "PLC8_CPU1214_DO_Vars".DO4.cMemory,
           iCounterIn := "PLC8_CPU1214_DO_Vars".DO4.iCounterIn,
           iCounterOut := "PLC8_CPU1214_DO_Vars".DO4.iCounterOut,
           xOutput => "PLC8_CPU1214_DO_Vars".DO4.xOutput);
   "DO8.01.04" := "PLC8_CPU1214_DO_Vars".DO4.xOutput;
END_REGION

REGION Network 21: DQ5
   RUNG wire#powerrail
      "DOvar"(iFuncSystem := "PLC8_CPU1214_DO_Vars".DO5.iFuncSystemID, iFuncVar := "PLC8_CPU1214_DO_Vars".DO5.iFuncVar, xOutput => "PLC8_CPU1214_DO_Vars".DO5.xInput)
   END_RUNG
   RUNG wire#powerrail
      "DOadv"(xInput := "PLC8_CPU1214_DO_Vars".DO5.xInput, xInversion := "PLC8_CPU1214_DO_Vars".DO5.xInversion, cMOA := "PLC8_CPU1214_DO_Vars".DO5.cMOA, xMemoryOut := "PLC8_CPU1214_DO_Vars".DO5.xMemoryOut, xMemoryIn := "PLC8_CPU1214_DO_Vars".DO5.xMemoryIn, cMemory := "PLC8_CPU1214_DO_Vars".DO5.cMemory, iCounterIn := "PLC8_CPU1214_DO_Vars".DO5.iCounterIn, iCounterOut := "PLC8_CPU1214_DO_Vars".DO5.iCounterOut, xOutput => "PLC8_CPU1214_DO_Vars".DO5.xOutput)
   END_RUNG
   RUNG wire#powerrail
      Contact( "PLC8_CPU1214_DO_Vars".DO5.xOutput )
      Coil( "DO8.01.05" )
   END_RUNG
   // the same network as SCL:
   "DOvar"(iFuncSystem := "PLC8_CPU1214_DO_Vars".DO5.iFuncSystemID,
           iFuncVar := "PLC8_CPU1214_DO_Vars".DO5.iFuncVar,
           xOutput => "PLC8_CPU1214_DO_Vars".DO5.xInput);
   "DOadv"(xInput := "PLC8_CPU1214_DO_Vars".DO5.xInput,
           xInversion := "PLC8_CPU1214_DO_Vars".DO5.xInversion,
           cMOA := "PLC8_CPU1214_DO_Vars".DO5.cMOA,
           xMemoryOut := "PLC8_CPU1214_DO_Vars".DO5.xMemoryOut,
           xMemoryIn := "PLC8_CPU1214_DO_Vars".DO5.xMemoryIn,
           cMemory := "PLC8_CPU1214_DO_Vars".DO5.cMemory,
           iCounterIn := "PLC8_CPU1214_DO_Vars".DO5.iCounterIn,
           iCounterOut := "PLC8_CPU1214_DO_Vars".DO5.iCounterOut,
           xOutput => "PLC8_CPU1214_DO_Vars".DO5.xOutput);
   "DO8.01.05" := "PLC8_CPU1214_DO_Vars".DO5.xOutput;
END_REGION

REGION Network 22: DQ6
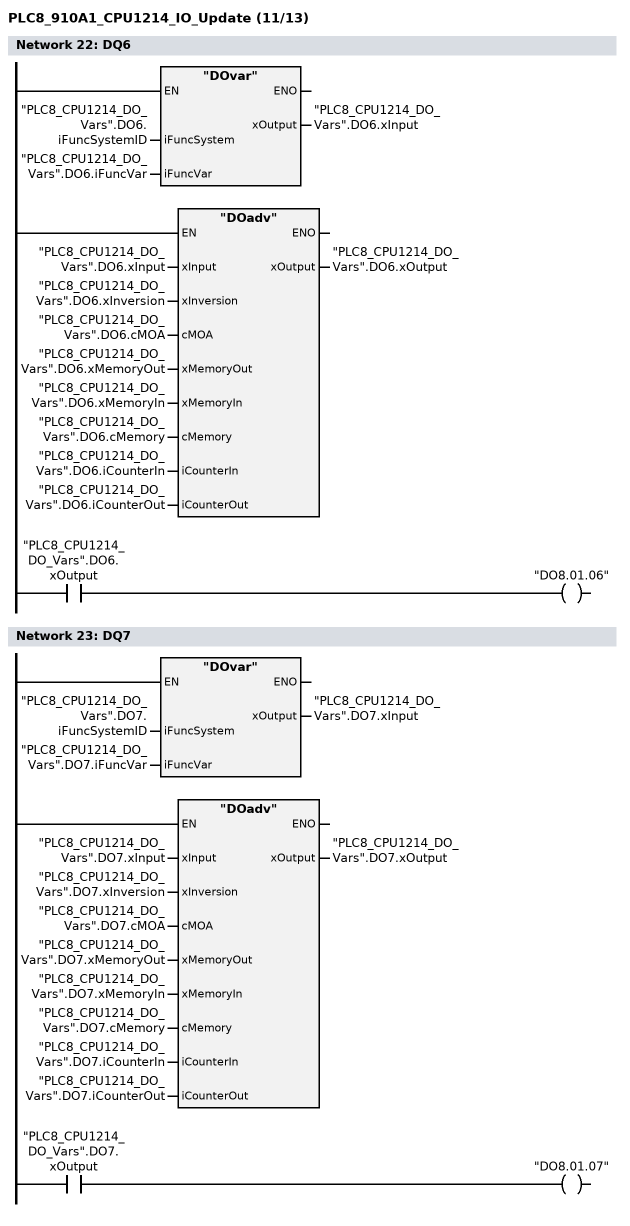
   RUNG wire#powerrail
      "DOvar"(iFuncSystem := "PLC8_CPU1214_DO_Vars".DO6.iFuncSystemID, iFuncVar := "PLC8_CPU1214_DO_Vars".DO6.iFuncVar, xOutput => "PLC8_CPU1214_DO_Vars".DO6.xInput)
   END_RUNG
   RUNG wire#powerrail
      "DOadv"(xInput := "PLC8_CPU1214_DO_Vars".DO6.xInput, xInversion := "PLC8_CPU1214_DO_Vars".DO6.xInversion, cMOA := "PLC8_CPU1214_DO_Vars".DO6.cMOA, xMemoryOut := "PLC8_CPU1214_DO_Vars".DO6.xMemoryOut, xMemoryIn := "PLC8_CPU1214_DO_Vars".DO6.xMemoryIn, cMemory := "PLC8_CPU1214_DO_Vars".DO6.cMemory, iCounterIn := "PLC8_CPU1214_DO_Vars".DO6.iCounterIn, iCounterOut := "PLC8_CPU1214_DO_Vars".DO6.iCounterOut, xOutput => "PLC8_CPU1214_DO_Vars".DO6.xOutput)
   END_RUNG
   RUNG wire#powerrail
      Contact( "PLC8_CPU1214_DO_Vars".DO6.xOutput )
      Coil( "DO8.01.06" )
   END_RUNG
   // the same network as SCL:
   "DOvar"(iFuncSystem := "PLC8_CPU1214_DO_Vars".DO6.iFuncSystemID,
           iFuncVar := "PLC8_CPU1214_DO_Vars".DO6.iFuncVar,
           xOutput => "PLC8_CPU1214_DO_Vars".DO6.xInput);
   "DOadv"(xInput := "PLC8_CPU1214_DO_Vars".DO6.xInput,
           xInversion := "PLC8_CPU1214_DO_Vars".DO6.xInversion,
           cMOA := "PLC8_CPU1214_DO_Vars".DO6.cMOA,
           xMemoryOut := "PLC8_CPU1214_DO_Vars".DO6.xMemoryOut,
           xMemoryIn := "PLC8_CPU1214_DO_Vars".DO6.xMemoryIn,
           cMemory := "PLC8_CPU1214_DO_Vars".DO6.cMemory,
           iCounterIn := "PLC8_CPU1214_DO_Vars".DO6.iCounterIn,
           iCounterOut := "PLC8_CPU1214_DO_Vars".DO6.iCounterOut,
           xOutput => "PLC8_CPU1214_DO_Vars".DO6.xOutput);
   "DO8.01.06" := "PLC8_CPU1214_DO_Vars".DO6.xOutput;
END_REGION

REGION Network 23: DQ7
   RUNG wire#powerrail
      "DOvar"(iFuncSystem := "PLC8_CPU1214_DO_Vars".DO7.iFuncSystemID, iFuncVar := "PLC8_CPU1214_DO_Vars".DO7.iFuncVar, xOutput => "PLC8_CPU1214_DO_Vars".DO7.xInput)
   END_RUNG
   RUNG wire#powerrail
      "DOadv"(xInput := "PLC8_CPU1214_DO_Vars".DO7.xInput, xInversion := "PLC8_CPU1214_DO_Vars".DO7.xInversion, cMOA := "PLC8_CPU1214_DO_Vars".DO7.cMOA, xMemoryOut := "PLC8_CPU1214_DO_Vars".DO7.xMemoryOut, xMemoryIn := "PLC8_CPU1214_DO_Vars".DO7.xMemoryIn, cMemory := "PLC8_CPU1214_DO_Vars".DO7.cMemory, iCounterIn := "PLC8_CPU1214_DO_Vars".DO7.iCounterIn, iCounterOut := "PLC8_CPU1214_DO_Vars".DO7.iCounterOut, xOutput => "PLC8_CPU1214_DO_Vars".DO7.xOutput)
   END_RUNG
   RUNG wire#powerrail
      Contact( "PLC8_CPU1214_DO_Vars".DO7.xOutput )
      Coil( "DO8.01.07" )
   END_RUNG
   // the same network as SCL:
   "DOvar"(iFuncSystem := "PLC8_CPU1214_DO_Vars".DO7.iFuncSystemID,
           iFuncVar := "PLC8_CPU1214_DO_Vars".DO7.iFuncVar,
           xOutput => "PLC8_CPU1214_DO_Vars".DO7.xInput);
   "DOadv"(xInput := "PLC8_CPU1214_DO_Vars".DO7.xInput,
           xInversion := "PLC8_CPU1214_DO_Vars".DO7.xInversion,
           cMOA := "PLC8_CPU1214_DO_Vars".DO7.cMOA,
           xMemoryOut := "PLC8_CPU1214_DO_Vars".DO7.xMemoryOut,
           xMemoryIn := "PLC8_CPU1214_DO_Vars".DO7.xMemoryIn,
           cMemory := "PLC8_CPU1214_DO_Vars".DO7.cMemory,
           iCounterIn := "PLC8_CPU1214_DO_Vars".DO7.iCounterIn,
           iCounterOut := "PLC8_CPU1214_DO_Vars".DO7.iCounterOut,
           xOutput => "PLC8_CPU1214_DO_Vars".DO7.xOutput);
   "DO8.01.07" := "PLC8_CPU1214_DO_Vars".DO7.xOutput;
END_REGION

REGION Network 24: DQ8
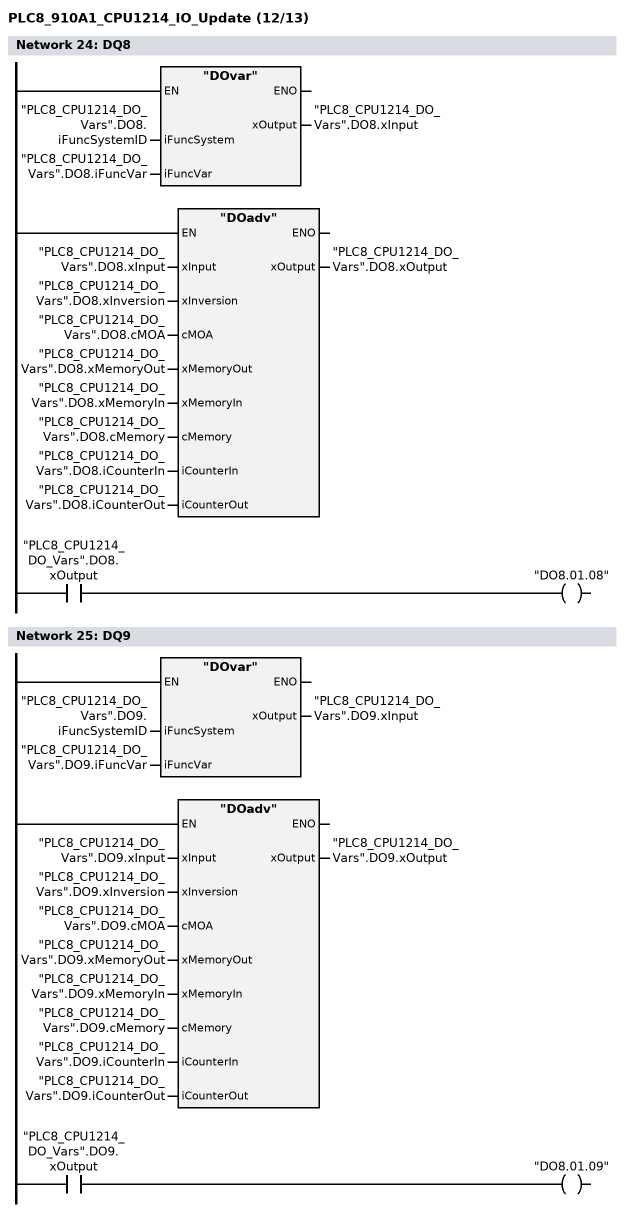
   RUNG wire#powerrail
      "DOvar"(iFuncSystem := "PLC8_CPU1214_DO_Vars".DO8.iFuncSystemID, iFuncVar := "PLC8_CPU1214_DO_Vars".DO8.iFuncVar, xOutput => "PLC8_CPU1214_DO_Vars".DO8.xInput)
   END_RUNG
   RUNG wire#powerrail
      "DOadv"(xInput := "PLC8_CPU1214_DO_Vars".DO8.xInput, xInversion := "PLC8_CPU1214_DO_Vars".DO8.xInversion, cMOA := "PLC8_CPU1214_DO_Vars".DO8.cMOA, xMemoryOut := "PLC8_CPU1214_DO_Vars".DO8.xMemoryOut, xMemoryIn := "PLC8_CPU1214_DO_Vars".DO8.xMemoryIn, cMemory := "PLC8_CPU1214_DO_Vars".DO8.cMemory, iCounterIn := "PLC8_CPU1214_DO_Vars".DO8.iCounterIn, iCounterOut := "PLC8_CPU1214_DO_Vars".DO8.iCounterOut, xOutput => "PLC8_CPU1214_DO_Vars".DO8.xOutput)
   END_RUNG
   RUNG wire#powerrail
      Contact( "PLC8_CPU1214_DO_Vars".DO8.xOutput )
      Coil( "DO8.01.08" )
   END_RUNG
   // the same network as SCL:
   "DOvar"(iFuncSystem := "PLC8_CPU1214_DO_Vars".DO8.iFuncSystemID,
           iFuncVar := "PLC8_CPU1214_DO_Vars".DO8.iFuncVar,
           xOutput => "PLC8_CPU1214_DO_Vars".DO8.xInput);
   "DOadv"(xInput := "PLC8_CPU1214_DO_Vars".DO8.xInput,
           xInversion := "PLC8_CPU1214_DO_Vars".DO8.xInversion,
           cMOA := "PLC8_CPU1214_DO_Vars".DO8.cMOA,
           xMemoryOut := "PLC8_CPU1214_DO_Vars".DO8.xMemoryOut,
           xMemoryIn := "PLC8_CPU1214_DO_Vars".DO8.xMemoryIn,
           cMemory := "PLC8_CPU1214_DO_Vars".DO8.cMemory,
           iCounterIn := "PLC8_CPU1214_DO_Vars".DO8.iCounterIn,
           iCounterOut := "PLC8_CPU1214_DO_Vars".DO8.iCounterOut,
           xOutput => "PLC8_CPU1214_DO_Vars".DO8.xOutput);
   "DO8.01.08" := "PLC8_CPU1214_DO_Vars".DO8.xOutput;
END_REGION

REGION Network 25: DQ9
   RUNG wire#powerrail
      "DOvar"(iFuncSystem := "PLC8_CPU1214_DO_Vars".DO9.iFuncSystemID, iFuncVar := "PLC8_CPU1214_DO_Vars".DO9.iFuncVar, xOutput => "PLC8_CPU1214_DO_Vars".DO9.xInput)
   END_RUNG
   RUNG wire#powerrail
      "DOadv"(xInput := "PLC8_CPU1214_DO_Vars".DO9.xInput, xInversion := "PLC8_CPU1214_DO_Vars".DO9.xInversion, cMOA := "PLC8_CPU1214_DO_Vars".DO9.cMOA, xMemoryOut := "PLC8_CPU1214_DO_Vars".DO9.xMemoryOut, xMemoryIn := "PLC8_CPU1214_DO_Vars".DO9.xMemoryIn, cMemory := "PLC8_CPU1214_DO_Vars".DO9.cMemory, iCounterIn := "PLC8_CPU1214_DO_Vars".DO9.iCounterIn, iCounterOut := "PLC8_CPU1214_DO_Vars".DO9.iCounterOut, xOutput => "PLC8_CPU1214_DO_Vars".DO9.xOutput)
   END_RUNG
   RUNG wire#powerrail
      Contact( "PLC8_CPU1214_DO_Vars".DO9.xOutput )
      Coil( "DO8.01.09" )
   END_RUNG
   // the same network as SCL:
   "DOvar"(iFuncSystem := "PLC8_CPU1214_DO_Vars".DO9.iFuncSystemID,
           iFuncVar := "PLC8_CPU1214_DO_Vars".DO9.iFuncVar,
           xOutput => "PLC8_CPU1214_DO_Vars".DO9.xInput);
   "DOadv"(xInput := "PLC8_CPU1214_DO_Vars".DO9.xInput,
           xInversion := "PLC8_CPU1214_DO_Vars".DO9.xInversion,
           cMOA := "PLC8_CPU1214_DO_Vars".DO9.cMOA,
           xMemoryOut := "PLC8_CPU1214_DO_Vars".DO9.xMemoryOut,
           xMemoryIn := "PLC8_CPU1214_DO_Vars".DO9.xMemoryIn,
           cMemory := "PLC8_CPU1214_DO_Vars".DO9.cMemory,
           iCounterIn := "PLC8_CPU1214_DO_Vars".DO9.iCounterIn,
           iCounterOut := "PLC8_CPU1214_DO_Vars".DO9.iCounterOut,
           xOutput => "PLC8_CPU1214_DO_Vars".DO9.xOutput);
   "DO8.01.09" := "PLC8_CPU1214_DO_Vars".DO9.xOutput;
END_REGION

REGION Network 26: DQ10
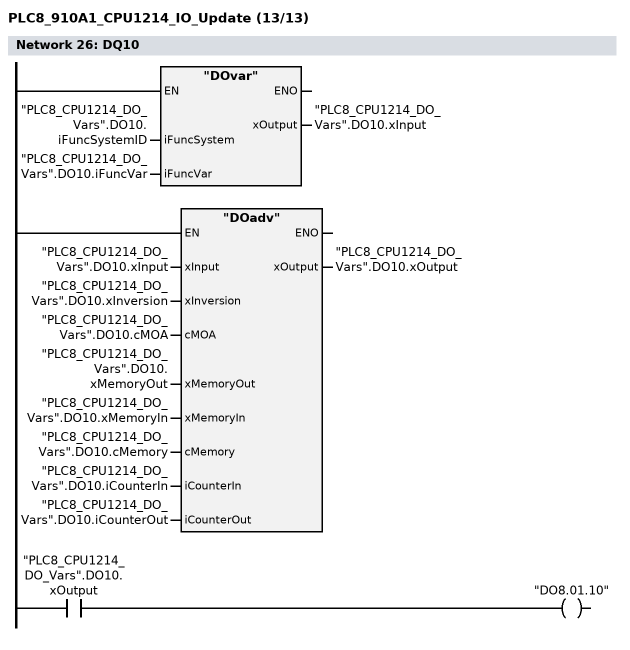
   RUNG wire#powerrail
      "DOvar"(iFuncSystem := "PLC8_CPU1214_DO_Vars".DO10.iFuncSystemID, iFuncVar := "PLC8_CPU1214_DO_Vars".DO10.iFuncVar, xOutput => "PLC8_CPU1214_DO_Vars".DO10.xInput)
   END_RUNG
   RUNG wire#powerrail
      "DOadv"(xInput := "PLC8_CPU1214_DO_Vars".DO10.xInput, xInversion := "PLC8_CPU1214_DO_Vars".DO10.xInversion, cMOA := "PLC8_CPU1214_DO_Vars".DO10.cMOA, xMemoryOut := "PLC8_CPU1214_DO_Vars".DO10.xMemoryOut, xMemoryIn := "PLC8_CPU1214_DO_Vars".DO10.xMemoryIn, cMemory := "PLC8_CPU1214_DO_Vars".DO10.cMemory, iCounterIn := "PLC8_CPU1214_DO_Vars".DO10.iCounterIn, iCounterOut := "PLC8_CPU1214_DO_Vars".DO10.iCounterOut, xOutput => "PLC8_CPU1214_DO_Vars".DO10.xOutput)
   END_RUNG
   RUNG wire#powerrail
      Contact( "PLC8_CPU1214_DO_Vars".DO10.xOutput )
      Coil( "DO8.01.10" )
   END_RUNG
   // the same network as SCL:
   "DOvar"(iFuncSystem := "PLC8_CPU1214_DO_Vars".DO10.iFuncSystemID,
           iFuncVar := "PLC8_CPU1214_DO_Vars".DO10.iFuncVar,
           xOutput => "PLC8_CPU1214_DO_Vars".DO10.xInput);
   "DOadv"(xInput := "PLC8_CPU1214_DO_Vars".DO10.xInput,
           xInversion := "PLC8_CPU1214_DO_Vars".DO10.xInversion,
           cMOA := "PLC8_CPU1214_DO_Vars".DO10.cMOA,
           xMemoryOut := "PLC8_CPU1214_DO_Vars".DO10.xMemoryOut,
           xMemoryIn := "PLC8_CPU1214_DO_Vars".DO10.xMemoryIn,
           cMemory := "PLC8_CPU1214_DO_Vars".DO10.cMemory,
           iCounterIn := "PLC8_CPU1214_DO_Vars".DO10.iCounterIn,
           iCounterOut := "PLC8_CPU1214_DO_Vars".DO10.iCounterOut,
           xOutput => "PLC8_CPU1214_DO_Vars".DO10.xOutput);
   "DO8.01.10" := "PLC8_CPU1214_DO_Vars".DO10.xOutput;
END_REGION
END_FUNCTION
